TYPE ST_P_GET_PARENT :
STRUCT
	ContainerId:			INT;
	Barcode:				INT;
END_STRUCT
END_TYPE

(* stored: Version 1.1.0.1, ProductVersion 3.1.4024.10
   DUT ST_P_GET_PARENT: Id {ddf1cd00-70e4-473e-8794-9e92033e8406} *)
